{attribute 'GeneratedUsingTerminal: CU2508--0000'}
{attribute addProperty BoxType "CU2508--0000"}
{attribute addProperty Id "EtcSlaveTerminalBaseInfoDataAT %I*InfoData_6F19DB2B2"}
{attribute addProperty CRC "2874840167"}
{attribute addProperty Size "2"}
TYPE CU2508_AB5A9467 EXTENDS EtcSlaveTerminalBase :
STRUCT
	{attribute addProperty Name "InfoData"}
	InfoData : InfoData_6F19DB2B;
END_STRUCT
END_TYPE

(* stored: Version 1.2.0.0, ProductVersion 3.1.4024.9
   DUT CU2508_AB5A9467: Id {030e95d9-6a16-4691-89cd-d48fc2b4b827} *)
